TYPE "MotorSAlr"
VERSION : 0.1
// Block: MotorSAlr
   STRUCT
      ThermalProtectionA : Bool;
      ThermalProtectionB : Bool;
      Feedback : Bool;
   END_STRUCT;

END_TYPE
